{attribute 'qualified_only'}
VAR_GLOBAL
	I AT %I* :Input;
	O AT %Q* :Output;
	Seq:FB_AutoSeq;
	Trunion:FB_Trunion;
END_VAR

(* stored: Version 1.1.0.1, ProductVersion 3.1.4024.16
   GVL Fixt1: Id {ec0d8970-4867-4559-8565-494de50d3377} *)
